% RSLogix 500 project WATER HEATER_BAK000.RSS, saved by version 9.00.00.04 %
PROJECT "UNTITLED"    % processor: MicroLogix 1400 %

PROGRAM FILES
  LAD 2   8 rungs

DATA FILES
  O0 OUTPUT  6 elements
  I1 INPUT  8 elements
  S2 STATUS  66 elements
  B3 BINARY  1 elements
  T4 TIMER  2 elements
  C5 COUNTER  2 elements
  R6 CONTROL  1 elements
  N7 INTEGER  1 elements
  F8 FLOAT  1 elements
  B9   10 elements
  B10   10 elements
  N14   10 elements
  N15   10 elements

LADDER 2
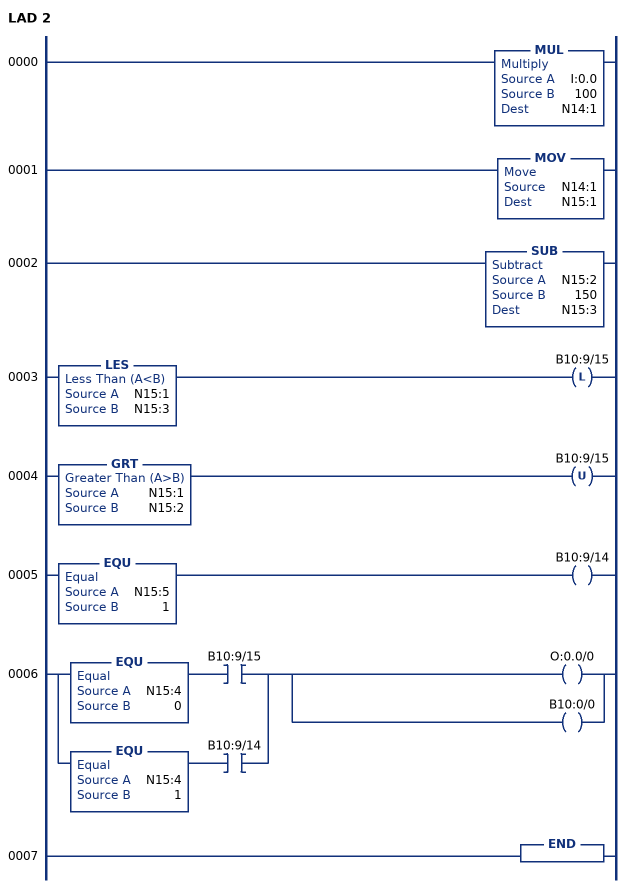
% Rung: 0 %
SOR MUL I:0.0 100 N14:1 EOR
% Rung: 1 %
SOR MOV N14:1 N15:1 EOR
% Rung: 2 %
SOR SUB N15:2 150 N15:3 EOR
% Rung: 3 %
SOR LES N15:1 N15:3 OTL B10:9/15 EOR
% Rung: 4 %
SOR GRT N15:1 N15:2 OTU B10:9/15 EOR
% Rung: 5 %
SOR EQU N15:5 1 OTE B10:9/14 EOR
% Rung: 6 %
SOR BST EQU N15:4 0 XIC B10:9/15 NXB EQU N15:4 1 XIC B10:9/14 BND BST OTE O:0.0/0 NXB OTE B10:0/0 BND EOR
% Rung: 7 %
SOR END EOR

DATA TABLE (non-zero values as saved)
DATA T4
% .PRE .ACC %
% T4:0 % 20 0
% T4:1 % 20 13
DATA C5
% .PRE .ACC %
% C5:0 % 100 51
% C5:1 % 0 10
DATA F8
% F8:0 % 4577.776
DATA B10
% B10:0 % 0X0000 0X0000 0X0000 0X0000 0X0000 0X0000 0X0000 0X0000 0X0000 0X8000
DATA N14
% N14:0 % 15000 0 0 0 0 0 0 0 0 0
DATA N15
% N15:0 % 0 0 4000 3850 1 0 8698 0 0 0
